// TIA Portal project "Progetto3" (V15.1)

(* hardware
DEVICE "S7-1200 station_1"  S7-1200 Station
   slot 0: "Telaio di montaggio_0"  S7-1200 Rack  Rack  V1.0
   slot 1: "PLC_1"  CPU 1214C DC/DC/DC  6ES7 214-1AG40-0XB0  V4.2
*)

// ===== PLC "PLC_1"  CPU 1214C DC/DC/DC =====

VAR_GLOBAL   // PLC tag table "Tabella delle variabili standard"
   "MS" AT %I0.0 : Bool;
   "MD" AT %I0.1 : Bool;
   "Mup" AT %I0.2 : Bool;
   "Mdown" AT %I0.3 : Bool;
   "L0" AT %M0.0 : Bool;
   "L1" AT %M0.1 : Bool;
   "V1" AT %M0.2 : Bool;
   "V2" AT %M0.3 : Bool;
   "stato1" AT %M0.4 : Bool;
   "stato2" AT %M0.5 : Bool;
END_VAR

DATA_BLOCK "variabili_stato"   // DB1
{ S7_Optimized_Access := 'TRUE' }
VERSION : 0.1
   VAR RETAIN
      Home : Bool := true;
   END_VAR
   VAR
      P1P2 : Bool;
      P2P1 : Bool;
      P1 : Bool;
      P2 : Bool;
      P1P0 : Bool;
      P0P1 : Bool;
   END_VAR
BEGIN
END_DATA_BLOCK

// folder: System blocks/Program resources

DATA_BLOCK "IEC_Timer_0_DB"   // DB2
{ S7_Optimized_Access := 'TRUE' }
AUTHOR : Simatic
FAMILY : IEC
NAME : IEC_TMR
VERSION : 1.0
// stored: InstanceOfName IEC_TIMER
"IEC_TIMER"
BEGIN
END_DATA_BLOCK

// folder: (top level)

ORGANIZATION_BLOCK "Main"   // OB1, LAD, ProgramCycle
TITLE = "Main Program Sweep (Cycle)"
{ S7_Optimized_Access := 'TRUE' }
VERSION : 0.1
   VAR_INPUT
      Initial_Call : Bool;   // Initial call of this OB
      Remanence : Bool;   // =True, if remanent data are available
   END_VAR
   VAR_TEMP   // added for the SCL form of the ladder/FBD networks
      _w1 : Bool;
   END_VAR
BEGIN

REGION Network 1
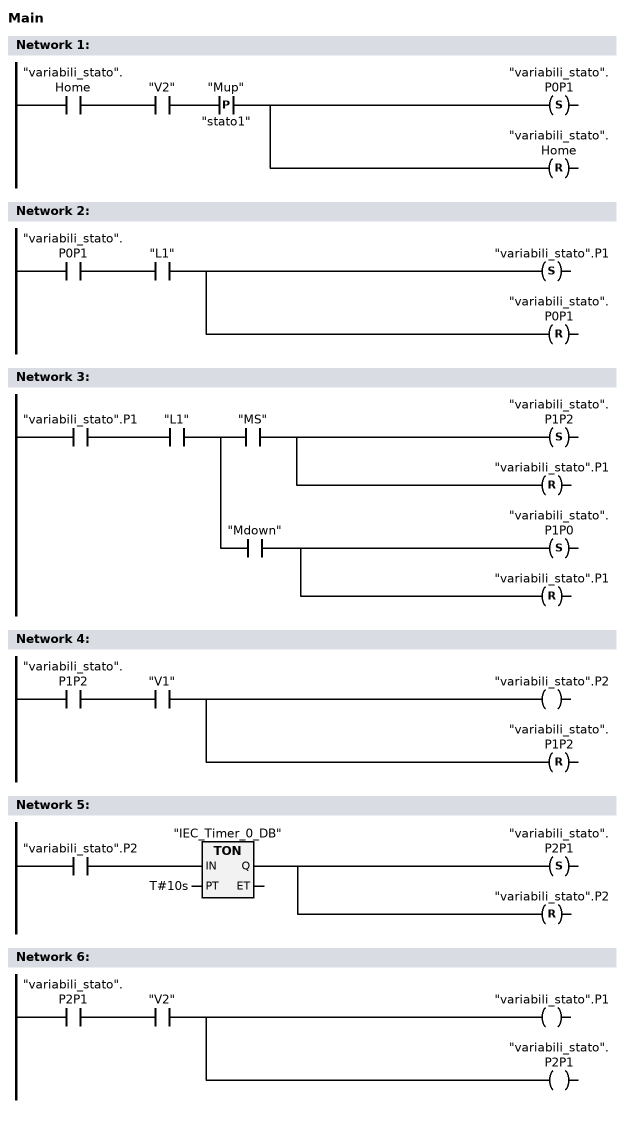
   RUNG wire#powerrail
      Contact( "variabili_stato".Home )
      Contact( "V2" )
      P_Contact(operand := "Mup", bit := "stato1")
      wire#w1
      S_Coil( "variabili_stato".P0P1 )
   END_RUNG
   RUNG wire#w1
      R_Coil( "variabili_stato".Home )
   END_RUNG
   // the same network as SCL:
   #_w1 := "variabili_stato".Home AND "V2" AND "Mup" AND NOT "stato1";   // rising edge of "Mup"
   "stato1" := "Mup";
   IF #_w1 THEN
       "variabili_stato".P0P1 := TRUE;
       "variabili_stato".Home := FALSE;
   END_IF;
END_REGION

REGION Network 2
   RUNG wire#powerrail
      Contact( "variabili_stato".P0P1 )
      Contact( "L1" )
      wire#w1
      S_Coil( "variabili_stato".P1 )
   END_RUNG
   RUNG wire#w1
      R_Coil( "variabili_stato".P0P1 )
   END_RUNG
   // the same network as SCL:
   IF "variabili_stato".P0P1 AND "L1" THEN
       "variabili_stato".P1 := TRUE;
       "variabili_stato".P0P1 := FALSE;
   END_IF;
END_REGION

REGION Network 3
   RUNG wire#powerrail
      Contact( "variabili_stato".P1 )
      Contact( "L1" )
      wire#w1
      Contact( "MS" )
      wire#w2
      S_Coil( "variabili_stato".P1P2 )
   END_RUNG
   RUNG wire#w2
      R_Coil( "variabili_stato".P1 )
   END_RUNG
   RUNG wire#w1
      Contact( "Mdown" )
      wire#w3
      S_Coil( "variabili_stato".P1P0 )
   END_RUNG
   RUNG wire#w3
      R_Coil( "variabili_stato".P1 )
   END_RUNG
   // the same network as SCL:
   #_w1 := "variabili_stato".P1 AND "L1";
   IF #_w1 AND "MS" THEN
       "variabili_stato".P1P2 := TRUE;
       "variabili_stato".P1 := FALSE;
   END_IF;
   IF #_w1 AND "Mdown" THEN
       "variabili_stato".P1P0 := TRUE;
       "variabili_stato".P1 := FALSE;
   END_IF;
END_REGION

REGION Network 4
   RUNG wire#powerrail
      Contact( "variabili_stato".P1P2 )
      Contact( "V1" )
      wire#w1
      Coil( "variabili_stato".P2 )
   END_RUNG
   RUNG wire#w1
      R_Coil( "variabili_stato".P1P2 )
   END_RUNG
   // the same network as SCL:
   "variabili_stato".P2 := "variabili_stato".P1P2 AND "V1";
   IF "variabili_stato".P2 THEN "variabili_stato".P1P2 := FALSE; END_IF;
END_REGION

REGION Network 5
   "IEC_Timer_0_DB".TON(IN := "variabili_stato".P2, PT := T#10s);
   IF "IEC_Timer_0_DB".Q THEN
       "variabili_stato".P2P1 := TRUE;
       "variabili_stato".P2 := FALSE;
   END_IF;
END_REGION

REGION Network 6
   RUNG wire#powerrail
      Contact( "variabili_stato".P2P1 )
      Contact( "V2" )
      wire#w1
      Coil( "variabili_stato".P1 )
   END_RUNG
   RUNG wire#w1
      Coil( "variabili_stato".P2P1 )
   END_RUNG
   // the same network as SCL:
   "variabili_stato".P1 := "variabili_stato".P2P1 AND "V2";
   "variabili_stato".P2P1 := "variabili_stato".P1;
END_REGION
END_ORGANIZATION_BLOCK